FUNCTION_BLOCK FeedforwardREAL (* Composite Function Block Type *)
  (* Standard: 61499-2 *)
  (* Version 0.0, 2018-09-24, 4DIAC-IDE, 4DIAC-Consortium *)
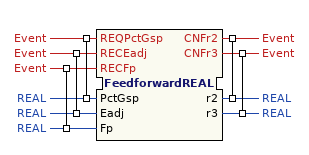
  EVENT_INPUT
    REQPctGsp WITH PctGsp;
    RECEadj WITH Eadj;
    RECFp WITH Fp;
  END_EVENT
  EVENT_OUTPUT
    CNFr2 WITH r2;
    CNFr3 WITH r3;
  END_EVENT
  VAR_INPUT
    PctGsp : REAL;
    Eadj : REAL;
    Fp : REAL;
  END_VAR
  VAR_OUTPUT
    r2 : REAL;
    r3 : REAL;
  END_VAR
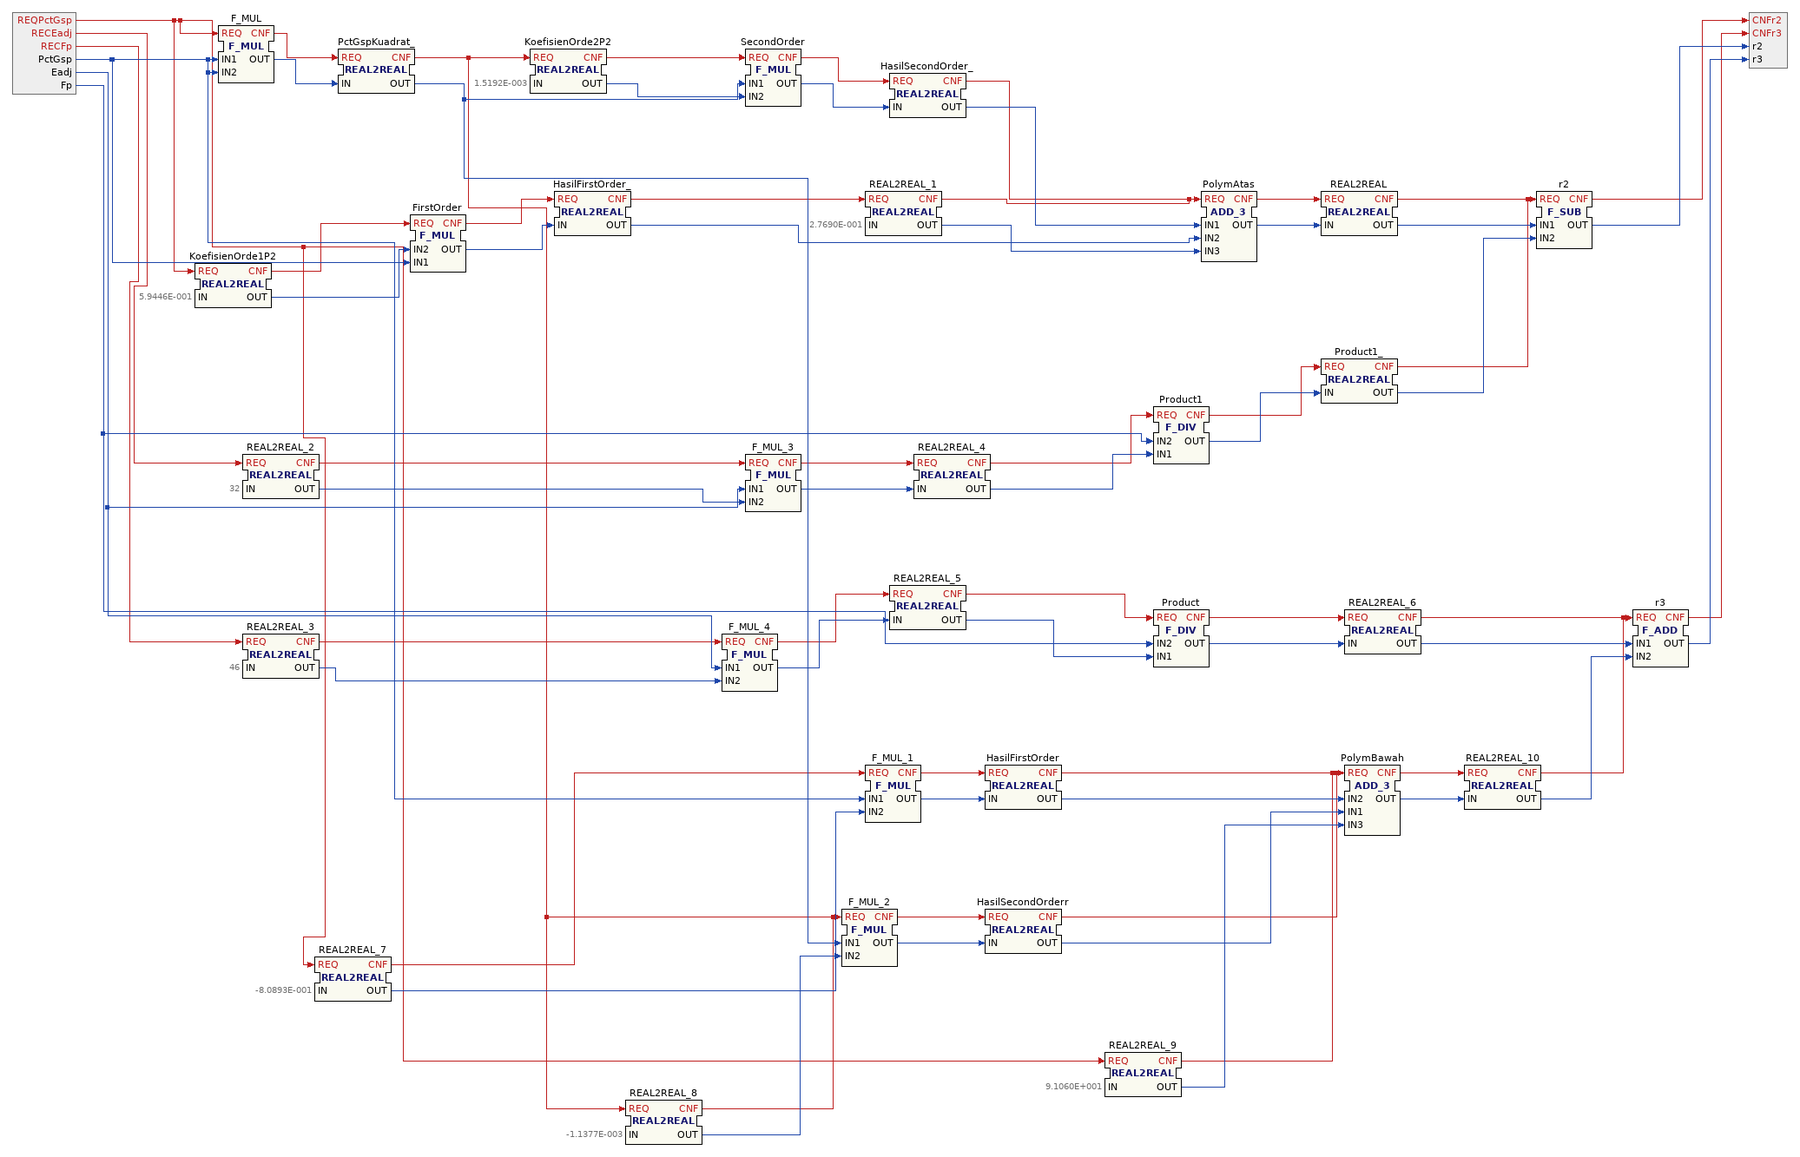
  FBS
    F_MUL : F_MUL;
    FirstOrder : F_MUL;
    PolymAtas : ADD_3;
    SecondOrder : F_MUL;
    PolymBawah : ADD_3;
    F_MUL_1 : F_MUL;
    F_MUL_2 : F_MUL;
    F_MUL_3 : F_MUL;
    F_MUL_4 : F_MUL;
    Product1 : F_DIV;
    Product : F_DIV;
    r2 : F_SUB;
    r3 : F_ADD;
    PctGspKuadrat_ : REAL2REAL;
    KoefisienOrde2P2 : REAL2REAL(IN := 1.5192E-003);
    HasilSecondOrder_ : REAL2REAL;
    KoefisienOrde1P2 : REAL2REAL(IN := 5.9446E-001);
    REAL2REAL_1 : REAL2REAL(IN := 2.7690E-001);
    HasilFirstOrder_ : REAL2REAL;
    REAL2REAL : REAL2REAL;
    Product1_ : REAL2REAL;
    REAL2REAL_2 : REAL2REAL(IN := 32);
    REAL2REAL_3 : REAL2REAL(IN := 46);
    REAL2REAL_4 : REAL2REAL;
    REAL2REAL_5 : REAL2REAL;
    REAL2REAL_6 : REAL2REAL;
    REAL2REAL_7 : REAL2REAL(IN := -8.0893E-001);
    HasilFirstOrder : REAL2REAL;
    REAL2REAL_8 : REAL2REAL(IN := -1.1377E-003);
    HasilSecondOrderr : REAL2REAL;
    REAL2REAL_9 : REAL2REAL(IN := 9.1060E+001);
    REAL2REAL_10 : REAL2REAL;
  END_FBS
  EVENT_CONNECTIONS
    F_MUL.CNF TO PctGspKuadrat_.REQ;
    PctGspKuadrat_.CNF TO F_MUL_2.REQ;
    PctGspKuadrat_.CNF TO KoefisienOrde2P2.REQ;
    KoefisienOrde2P2.CNF TO SecondOrder.REQ;
    SecondOrder.CNF TO HasilSecondOrder_.REQ;
    HasilSecondOrder_.CNF TO PolymAtas.REQ;
    KoefisienOrde1P2.CNF TO FirstOrder.REQ;
    FirstOrder.CNF TO HasilFirstOrder_.REQ;
    REAL2REAL_1.CNF TO PolymAtas.REQ;
    HasilFirstOrder_.CNF TO REAL2REAL_1.REQ;
    PolymAtas.CNF TO REAL2REAL.REQ;
    REAL2REAL.CNF TO r2.REQ;
    Product1_.CNF TO r2.REQ;
    Product1.CNF TO Product1_.REQ;
    REQPctGsp TO KoefisienOrde1P2.REQ;
    REQPctGsp TO F_MUL.REQ;
    r2.CNF TO CNFr2;
    RECEadj TO REAL2REAL_2.REQ;
    REAL2REAL_2.CNF TO F_MUL_3.REQ;
    RECFp TO REAL2REAL_3.REQ;
    REAL2REAL_3.CNF TO F_MUL_4.REQ;
    REAL2REAL_4.CNF TO Product1.REQ;
    F_MUL_3.CNF TO REAL2REAL_4.REQ;
    F_MUL_4.CNF TO REAL2REAL_5.REQ;
    REAL2REAL_5.CNF TO Product.REQ;
    Product.CNF TO REAL2REAL_6.REQ;
    REAL2REAL_6.CNF TO r3.REQ;
    REQPctGsp TO REAL2REAL_7.REQ;
    REAL2REAL_7.CNF TO F_MUL_1.REQ;
    F_MUL_1.CNF TO HasilFirstOrder.REQ;
    HasilFirstOrder.CNF TO PolymBawah.REQ;
    PctGspKuadrat_.CNF TO REAL2REAL_8.REQ;
    REAL2REAL_8.CNF TO F_MUL_2.REQ;
    F_MUL_2.CNF TO HasilSecondOrderr.REQ;
    HasilSecondOrderr.CNF TO PolymBawah.REQ;
    REQPctGsp TO REAL2REAL_9.REQ;
    REAL2REAL_9.CNF TO PolymBawah.REQ;
    REAL2REAL_10.CNF TO r3.REQ;
    PolymBawah.CNF TO REAL2REAL_10.REQ;
    r3.CNF TO CNFr3;
  END_CONNECTIONS
  DATA_CONNECTIONS
    F_MUL.OUT TO PctGspKuadrat_.IN;
    PctGspKuadrat_.OUT TO F_MUL_2.IN1;
    PctGspKuadrat_.OUT TO SecondOrder.IN1;
    KoefisienOrde2P2.OUT TO SecondOrder.IN2;
    SecondOrder.OUT TO HasilSecondOrder_.IN;
    HasilSecondOrder_.OUT TO PolymAtas.IN1;
    KoefisienOrde1P2.OUT TO FirstOrder.IN2;
    FirstOrder.OUT TO HasilFirstOrder_.IN;
    HasilFirstOrder_.OUT TO PolymAtas.IN2;
    REAL2REAL_1.OUT TO PolymAtas.IN3;
    PolymAtas.OUT TO REAL2REAL.IN;
    REAL2REAL.OUT TO r2.IN1;
    Product1_.OUT TO r2.IN2;
    Product1.OUT TO Product1_.IN;
    PctGsp TO F_MUL.IN1;
    PctGsp TO F_MUL.IN2;
    PctGsp TO FirstOrder.IN1;
    PctGsp TO F_MUL_1.IN1;
    r2.OUT TO r2;
    Eadj TO F_MUL_4.IN1;
    Eadj TO F_MUL_3.IN1;
    REAL2REAL_2.OUT TO F_MUL_3.IN2;
    Fp TO Product.IN2;
    Fp TO Product1.IN2;
    REAL2REAL_3.OUT TO F_MUL_4.IN2;
    F_MUL_3.OUT TO REAL2REAL_4.IN;
    REAL2REAL_4.OUT TO Product1.IN1;
    F_MUL_4.OUT TO REAL2REAL_5.IN;
    REAL2REAL_5.OUT TO Product.IN1;
    Product.OUT TO REAL2REAL_6.IN;
    REAL2REAL_6.OUT TO r3.IN1;
    REAL2REAL_7.OUT TO F_MUL_1.IN2;
    F_MUL_1.OUT TO HasilFirstOrder.IN;
    HasilFirstOrder.OUT TO PolymBawah.IN2;
    REAL2REAL_8.OUT TO F_MUL_2.IN2;
    F_MUL_2.OUT TO HasilSecondOrderr.IN;
    HasilSecondOrderr.OUT TO PolymBawah.IN1;
    REAL2REAL_9.OUT TO PolymBawah.IN3;
    PolymBawah.OUT TO REAL2REAL_10.IN;
    REAL2REAL_10.OUT TO r3.IN2;
    r3.OUT TO r3;
  END_CONNECTIONS
END_FUNCTION_BLOCK
